FUNCTION_BLOCK EventLogger
VAR
	EventBuffer : ARRAY[1..MAXIMUM_SIZE_OF_EVENT_BUFFER] OF ST_Event;
	CurrentEventBufferIndex : INT := 0;
	
	_PersistentEventStorage : I_PersistentEventStorage;
END_VAR
VAR CONSTANT
	MAXIMUM_SIZE_OF_EVENT_BUFFER : INT := 100;
END_VAR

(* Returns TRUE if add succesful and FALSe if buffer is full *)
METHOD PUBLIC AddEvent : BOOL
VAR_INPUT
	eEventType : E_EventType;
	eEventSeverity : TcEventSeverity;
	nEventIdentity : UDINT;
	sEventText : STRING(255);
END_VAR
IF NOT IsEventBufferFull() THEN
	CurrentEventBufferIndex := CurrentEventBufferIndex + 1;
	eventbuffer[CurrentEventBufferIndex].eEventType := eEventType;
	eventbuffer[CurrentEventBufferIndex].eEventSeverity := eEventSeverity;
	eventbuffer[CurrentEventBufferIndex].nEventIdentity := nEventIdentity;
	eventbuffer[CurrentEventBufferIndex].sEventText := sEventText;
	UpdateEventTimestampWithSystemTime(stEvent := eventbuffer[CurrentEventBufferIndex]);
	AddEvent := TRUE;
ELSE
	AddEvent := FALSE;
END_IF

// Here we wan't to store the event persistently
_PersistentEventStorage.StoreEvent(stEvent := eventbuffer[CurrentEventBufferIndex]);
END_METHOD

METHOD FB_init : BOOL
VAR_INPUT
	bInitRetains : BOOL; // if TRUE, the retain variables are initialized (warm start / cold start)
	bInCopyCode : BOOL;  // if TRUE, the instance afterwards gets moved into the copy code (online change)
	iPersistentEventStorage : I_PersistentEventStorage;
END_VAR
_PersistentEventStorage := iPersistentEventStorage;
END_METHOD

METHOD PRIVATE IsEventBufferFull : BOOL
IsEventBufferFull := (CurrentEventBufferIndex + 1) > MAXIMUM_SIZE_OF_EVENT_BUFFER;
END_METHOD

END_FUNCTION_BLOCK

(* stored: Version 1.1.0.1, ProductVersion 3.1.4024.12
   POU EventLogger: Id {6e5f6654-9ffc-428b-845c-49dda0471b4b}, SpecialFunc None
   Method AddEvent: Id {36c01e8a-7b53-4398-a896-23c33bd706ab}
   Method FB_init: Id {77818cd6-c496-4ead-807f-1754b8913861}
   Method IsEventBufferFull: Id {d68c9b9e-6636-4f39-826d-0dcc3fee0f8e} *)
